// TIA Portal V19 export
DATA_BLOCK "A0301_Spintore_Lat_PERS"   // DB35
// stored: MemoryReserve 100
   VAR RETAIN
      Spin_Lat_1 : Struct
         Par { S7_SetPoint := 'True'} : "Analogic_SensorManagement_Par";
         Data : Struct
            Sens { S7_SetPoint := 'True'} : "Analogic_SensorManagement_Data";
            HMI { ExternalAccessible := 'False'; ExternalVisible := 'False'; ExternalWritable := 'False'} : "HMI_Preset";
         END_STRUCT;
         Par_Mach { S7_SetPoint := 'True'} : "A0301_Mach_Sens_Par";
      END_STRUCT;
      Spin_Lat_2 : Struct
         Par : "Analogic_SensorManagement_Par";
         Data : Struct
            Sens { S7_SetPoint := 'True'} : "Analogic_SensorManagement_Data";
            HMI : "HMI_Preset";
         END_STRUCT;
         Par_Mach : "A0301_Mach_Sens_Par";
      END_STRUCT;
   END_VAR
BEGIN
   Spin_Lat_1.Par.Enable := TRUE;   // 1= Enable / 0 Disable
   Spin_Lat_1.Par.RangeLow := 260.0;   // Corsa minima pistone
   Spin_Lat_1.Par.RangeHigh := 60.0;   // Corsa massima pistone
   Spin_Lat_1.Data.Sens.OffsetValue := 5.88212585449219;   // Valore aggiunto o sottratto a Out.ScaleValue
   Spin_Lat_1.Data.Sens.OffsetValid := TRUE;   // Stato di ritorno del valore offset
   Spin_Lat_1.Data.HMI.Button := FALSE;
   Spin_Lat_1.Data.HMI.Value := 260.0;
   Spin_Lat_1.Data.HMI.Feedback := 260.029876708984;
   Spin_Lat_1.Par_Mach.Tol_Work := 180.0;
   Spin_Lat_1.Par_Mach.WorkTime_SensDisable := T#100MS;
   Spin_Lat_2.Par.Enable := TRUE;   // 1= Enable / 0 Disable
   Spin_Lat_2.Par.RangeLow := 260.0;   // Corsa minima pistone
   Spin_Lat_2.Par.RangeHigh := 60.0;   // Corsa massima pistone
   Spin_Lat_2.Data.Sens.OffsetValue := 6.43084716796875;   // Valore aggiunto o sottratto a Out.ScaleValue
   Spin_Lat_2.Data.Sens.OffsetValid := TRUE;   // Stato di ritorno del valore offset
   Spin_Lat_2.Data.HMI.Button := FALSE;
   Spin_Lat_2.Data.HMI.Value := 260.0;
   Spin_Lat_2.Data.HMI.Feedback := 260.0;
   Spin_Lat_2.Par_Mach.Tol_Work := 180.0;
   Spin_Lat_2.Par_Mach.WorkTime_SensDisable := T#100MS;
END_DATA_BLOCK
